// TIA Portal V20 export
FUNCTION_BLOCK "F-FB_Axis"   // FB130, F_LAD
{ S7_Optimized_Access := 'TRUE' }
// stored: AutoNumber false
   VAR
      LDrvSafe_SinaTlg903StatusAxis01_X : "LDrvSafe_SinaTlg903Status";
      LDrvSafe_SinaTlg903StatusAxis02_Y : "LDrvSafe_SinaTlg903Status";
      LDrvSafe_SinaTlg903StatusAxis03_ZM : "LDrvSafe_SinaTlg903Status";
      LDrvSafe_SinaTlg903StatusAxis04_B : "LDrvSafe_SinaTlg903Status";
      LDrvSafe_SinaTlg903StatusAxis05_U1 : "LDrvSafe_SinaTlg903Status";
      LDrvSafe_SinaTlg903StatusAxis06_U2 : "LDrvSafe_SinaTlg903Status";
      LDrvSafe_SinaTlg903StatusAxis07_V : "LDrvSafe_SinaTlg903Status";
      LDrvSafe_SinaTlg903StatusAxis08_W : "LDrvSafe_SinaTlg903Status";
      LDrvSafe_SinaTlg903StatusAxis09_ZL : "LDrvSafe_SinaTlg903Status";
      LDrvSafe_SinaTlg903ControlAxis01_X : "LDrvSafe_SinaTlg903Control";
      LDrvSafe_SinaTlg903ControlAxis02_Y : "LDrvSafe_SinaTlg903Control";
      LDrvSafe_SinaTlg903ControlAxis03_ZM : "LDrvSafe_SinaTlg903Control";
      LDrvSafe_SinaTlg903ControlAxis04_B : "LDrvSafe_SinaTlg903Control";
      LDrvSafe_SinaTlg903ControlAxis05_U1 : "LDrvSafe_SinaTlg903Control";
      LDrvSafe_SinaTlg903ControlAxis06_U2 : "LDrvSafe_SinaTlg903Control";
      LDrvSafe_SinaTlg903ControlAxis07_V : "LDrvSafe_SinaTlg903Control";
      LDrvSafe_SinaTlg903ControlAxis08_W : "LDrvSafe_SinaTlg903Control";
      LDrvSafe_SinaTlg903ControlAxis09_ZL : "LDrvSafe_SinaTlg903Control";
   END_VAR
   VAR_TEMP
      tEnable_Axis_Move : Bool;
   END_VAR
BEGIN

REGION Network 1: Enable Axis Move
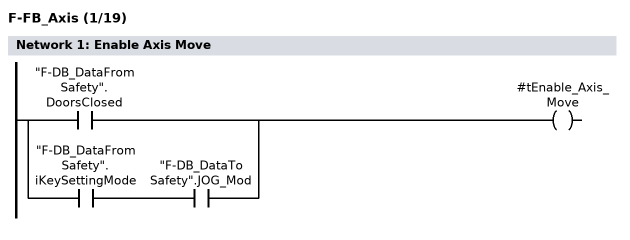
   RUNG wire#powerrail
      Contact( "F-DB_DataFromSafety".DoorsClosed )
      wire#w1
      Coil( #tEnable_Axis_Move )
   END_RUNG
   RUNG wire#powerrail
      Contact( "F-DB_DataFromSafety".iKeySettingMode )
      Contact( "F-DB_DataToSafety".JOG_Mod )
   END_RUNG wire#w1
   // the same network as SCL:
   #tEnable_Axis_Move := "F-DB_DataFromSafety".DoorsClosed OR ("F-DB_DataFromSafety".iKeySettingMode AND "F-DB_DataToSafety".JOG_Mod);
END_REGION

REGION Network 2: Axis01_X Status
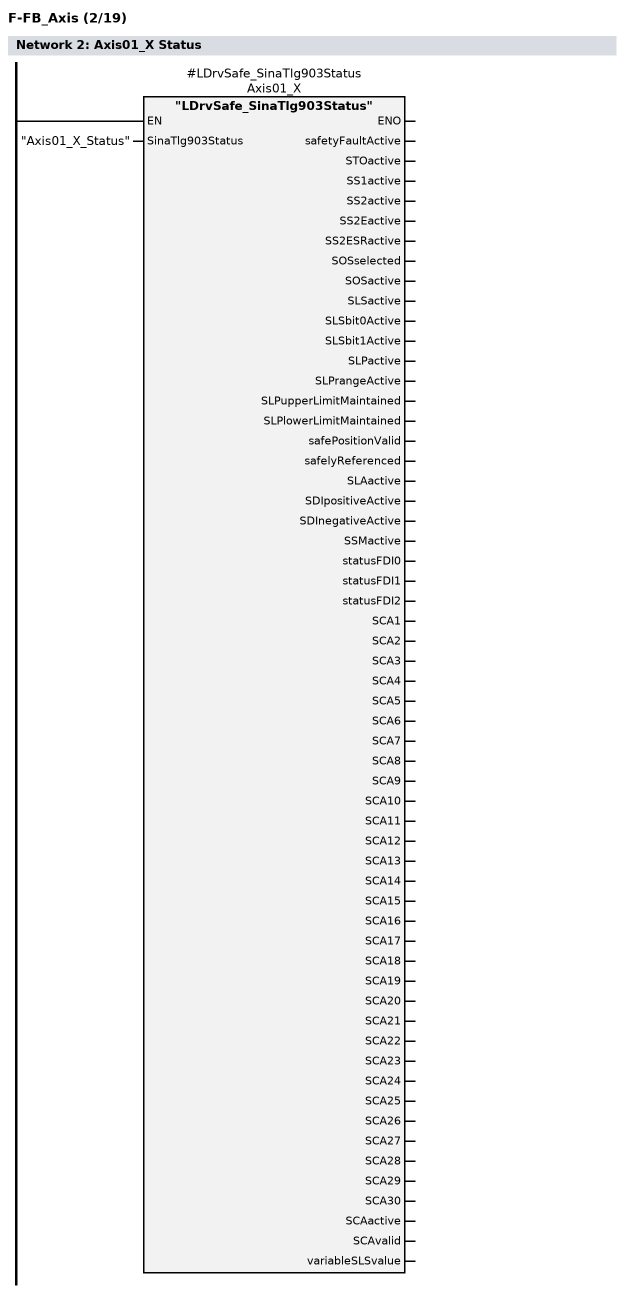
   RUNG wire#powerrail
      #LDrvSafe_SinaTlg903StatusAxis01_X(SinaTlg903Status := "Axis01_X_Status", safetyFaultActive =>, STOactive =>, SS1active =>, SS2active =>, SS2Eactive =>, SS2ESRactive =>, SOSselected =>, SOSactive =>, SLSactive =>, SLSbit0Active =>, SLSbit1Active =>, SLPactive =>, SLPrangeActive =>, SLPupperLimitMaintained =>, SLPlowerLimitMaintained =>, safePositionValid =>, safelyReferenced =>, SLAactive =>, SDIpositiveActive =>, SDInegativeActive =>, SSMactive =>, statusFDI0 =>, statusFDI1 =>, statusFDI2 =>, SCA1 =>, SCA2 =>, SCA3 =>, SCA4 =>, SCA5 =>, SCA6 =>, SCA7 =>, SCA8 =>, SCA9 =>, SCA10 =>, SCA11 =>, SCA12 =>, SCA13 =>, SCA14 =>, SCA15 =>, SCA16 =>, SCA17 =>, SCA18 =>, SCA19 =>, SCA20 =>, SCA21 =>, SCA22 =>, SCA23 =>, SCA24 =>, SCA25 =>, SCA26 =>, SCA27 =>, SCA28 =>, SCA29 =>, SCA30 =>, SCAactive =>, SCAvalid =>, variableSLSvalue =>)
   END_RUNG
   // the same network as SCL:
   #LDrvSafe_SinaTlg903StatusAxis01_X(SinaTlg903Status := "Axis01_X_Status");   // "LDrvSafe_SinaTlg903Status"
END_REGION

REGION Network 3: Axis01_X Control
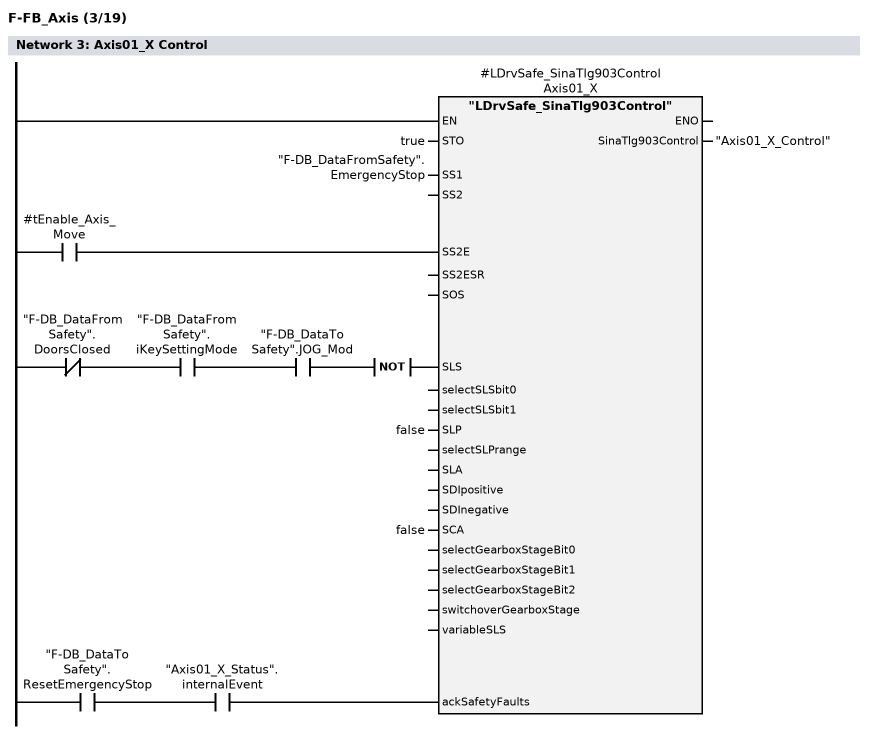
   RUNG wire#powerrail
      #LDrvSafe_SinaTlg903ControlAxis01_X(SS2E := wire#w1, SLS := wire#w2, ackSafetyFaults := wire#w3, STO := true, SS1 := "F-DB_DataFromSafety".EmergencyStop, SS2 :=, SS2ESR :=, SOS :=, selectSLSbit0 :=, selectSLSbit1 :=, SLP := false, selectSLPrange :=, SLA :=, SDIpositive :=, SDInegative :=, SCA := false, selectGearboxStageBit0 :=, selectGearboxStageBit1 :=, selectGearboxStageBit2 :=, switchoverGearboxStage :=, variableSLS :=, SinaTlg903Control => "Axis01_X_Control")
   END_RUNG
   RUNG wire#powerrail
      Contact( #tEnable_Axis_Move )
   END_RUNG wire#w1
   RUNG wire#powerrail
      I_Contact( "F-DB_DataFromSafety".DoorsClosed )
      Contact( "F-DB_DataFromSafety".iKeySettingMode )
      Contact( "F-DB_DataToSafety".JOG_Mod )
      Not()
   END_RUNG wire#w2
   RUNG wire#powerrail
      Contact( "F-DB_DataToSafety".ResetEmergencyStop )
      Contact( "Axis01_X_Status".internalEvent )
   END_RUNG wire#w3
   // the same network as SCL:
   #LDrvSafe_SinaTlg903ControlAxis01_X(STO := true,   // "LDrvSafe_SinaTlg903Control"
                           SS1 := "F-DB_DataFromSafety".EmergencyStop,
                           SS2E := #tEnable_Axis_Move,
                           SLS := NOT (NOT "F-DB_DataFromSafety".DoorsClosed AND "F-DB_DataFromSafety".iKeySettingMode AND "F-DB_DataToSafety".JOG_Mod),
                           SLP := false,
                           SCA := false,
                           ackSafetyFaults := "F-DB_DataToSafety".ResetEmergencyStop AND "Axis01_X_Status".internalEvent,
                           SinaTlg903Control => "Axis01_X_Control");
END_REGION

REGION Network 4: Axis02_Y Status
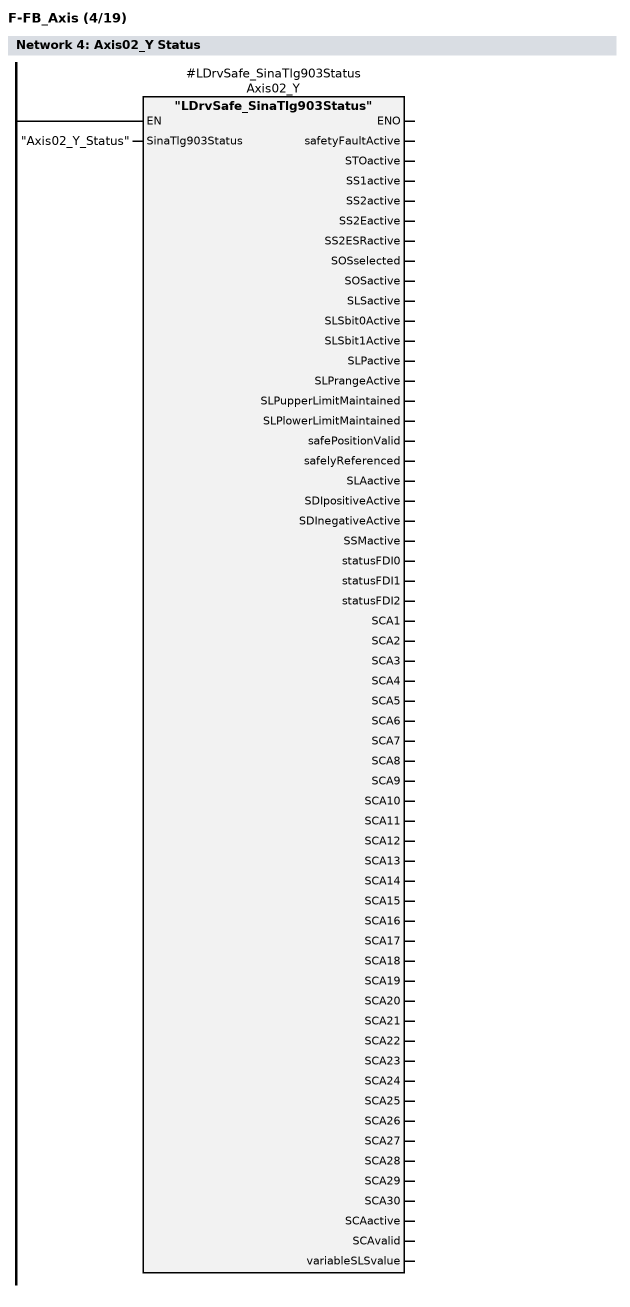
   RUNG wire#powerrail
      #LDrvSafe_SinaTlg903StatusAxis02_Y(SinaTlg903Status := "Axis02_Y_Status", safetyFaultActive =>, STOactive =>, SS1active =>, SS2active =>, SS2Eactive =>, SS2ESRactive =>, SOSselected =>, SOSactive =>, SLSactive =>, SLSbit0Active =>, SLSbit1Active =>, SLPactive =>, SLPrangeActive =>, SLPupperLimitMaintained =>, SLPlowerLimitMaintained =>, safePositionValid =>, safelyReferenced =>, SLAactive =>, SDIpositiveActive =>, SDInegativeActive =>, SSMactive =>, statusFDI0 =>, statusFDI1 =>, statusFDI2 =>, SCA1 =>, SCA2 =>, SCA3 =>, SCA4 =>, SCA5 =>, SCA6 =>, SCA7 =>, SCA8 =>, SCA9 =>, SCA10 =>, SCA11 =>, SCA12 =>, SCA13 =>, SCA14 =>, SCA15 =>, SCA16 =>, SCA17 =>, SCA18 =>, SCA19 =>, SCA20 =>, SCA21 =>, SCA22 =>, SCA23 =>, SCA24 =>, SCA25 =>, SCA26 =>, SCA27 =>, SCA28 =>, SCA29 =>, SCA30 =>, SCAactive =>, SCAvalid =>, variableSLSvalue =>)
   END_RUNG
   // the same network as SCL:
   #LDrvSafe_SinaTlg903StatusAxis02_Y(SinaTlg903Status := "Axis02_Y_Status");   // "LDrvSafe_SinaTlg903Status"
END_REGION

REGION Network 5: Axis02_Y Control
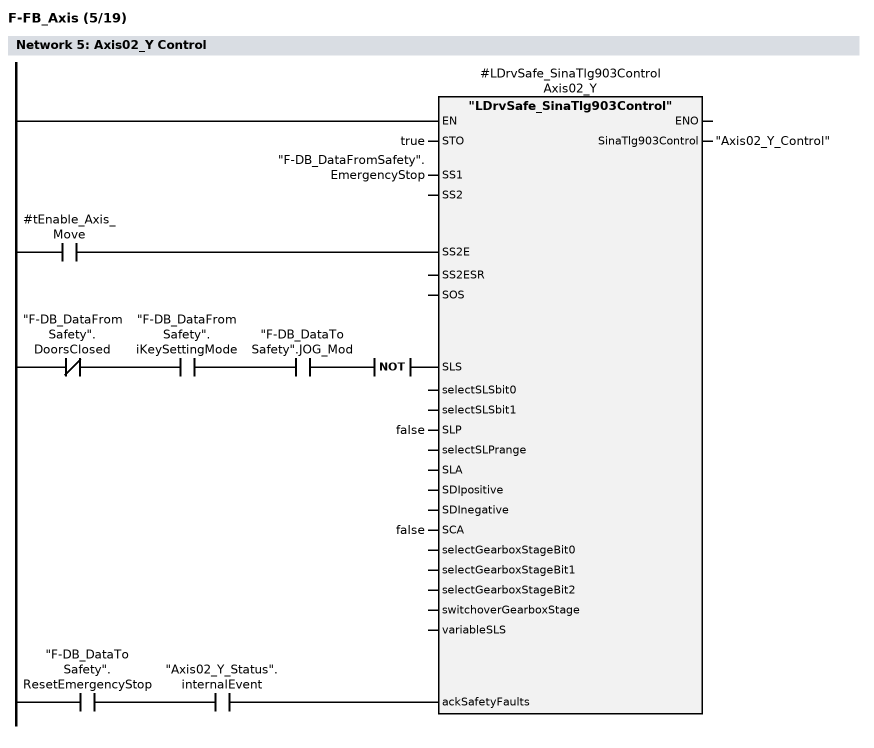
   RUNG wire#powerrail
      #LDrvSafe_SinaTlg903ControlAxis02_Y(SS2E := wire#w1, SLS := wire#w2, ackSafetyFaults := wire#w3, STO := true, SS1 := "F-DB_DataFromSafety".EmergencyStop, SS2 :=, SS2ESR :=, SOS :=, selectSLSbit0 :=, selectSLSbit1 :=, SLP := false, selectSLPrange :=, SLA :=, SDIpositive :=, SDInegative :=, SCA := false, selectGearboxStageBit0 :=, selectGearboxStageBit1 :=, selectGearboxStageBit2 :=, switchoverGearboxStage :=, variableSLS :=, SinaTlg903Control => "Axis02_Y_Control")
   END_RUNG
   RUNG wire#powerrail
      Contact( #tEnable_Axis_Move )
   END_RUNG wire#w1
   RUNG wire#powerrail
      I_Contact( "F-DB_DataFromSafety".DoorsClosed )
      Contact( "F-DB_DataFromSafety".iKeySettingMode )
      Contact( "F-DB_DataToSafety".JOG_Mod )
      Not()
   END_RUNG wire#w2
   RUNG wire#powerrail
      Contact( "F-DB_DataToSafety".ResetEmergencyStop )
      Contact( "Axis02_Y_Status".internalEvent )
   END_RUNG wire#w3
   // the same network as SCL:
   #LDrvSafe_SinaTlg903ControlAxis02_Y(STO := true,   // "LDrvSafe_SinaTlg903Control"
                           SS1 := "F-DB_DataFromSafety".EmergencyStop,
                           SS2E := #tEnable_Axis_Move,
                           SLS := NOT (NOT "F-DB_DataFromSafety".DoorsClosed AND "F-DB_DataFromSafety".iKeySettingMode AND "F-DB_DataToSafety".JOG_Mod),
                           SLP := false,
                           SCA := false,
                           ackSafetyFaults := "F-DB_DataToSafety".ResetEmergencyStop AND "Axis02_Y_Status".internalEvent,
                           SinaTlg903Control => "Axis02_Y_Control");
END_REGION

REGION Network 6: Axis03_ZM Status
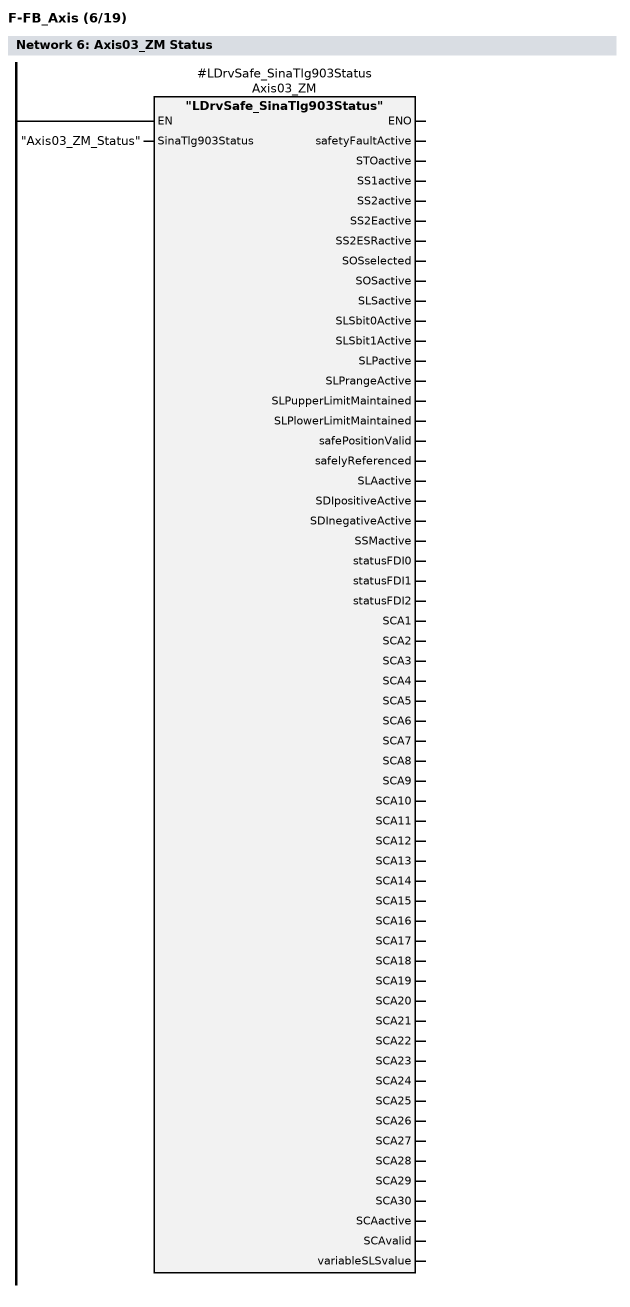
   RUNG wire#powerrail
      #LDrvSafe_SinaTlg903StatusAxis03_ZM(SinaTlg903Status := "Axis03_ZM_Status", safetyFaultActive =>, STOactive =>, SS1active =>, SS2active =>, SS2Eactive =>, SS2ESRactive =>, SOSselected =>, SOSactive =>, SLSactive =>, SLSbit0Active =>, SLSbit1Active =>, SLPactive =>, SLPrangeActive =>, SLPupperLimitMaintained =>, SLPlowerLimitMaintained =>, safePositionValid =>, safelyReferenced =>, SLAactive =>, SDIpositiveActive =>, SDInegativeActive =>, SSMactive =>, statusFDI0 =>, statusFDI1 =>, statusFDI2 =>, SCA1 =>, SCA2 =>, SCA3 =>, SCA4 =>, SCA5 =>, SCA6 =>, SCA7 =>, SCA8 =>, SCA9 =>, SCA10 =>, SCA11 =>, SCA12 =>, SCA13 =>, SCA14 =>, SCA15 =>, SCA16 =>, SCA17 =>, SCA18 =>, SCA19 =>, SCA20 =>, SCA21 =>, SCA22 =>, SCA23 =>, SCA24 =>, SCA25 =>, SCA26 =>, SCA27 =>, SCA28 =>, SCA29 =>, SCA30 =>, SCAactive =>, SCAvalid =>, variableSLSvalue =>)
   END_RUNG
   // the same network as SCL:
   #LDrvSafe_SinaTlg903StatusAxis03_ZM(SinaTlg903Status := "Axis03_ZM_Status");   // "LDrvSafe_SinaTlg903Status"
END_REGION

REGION Network 7: Axis03_ZM Control
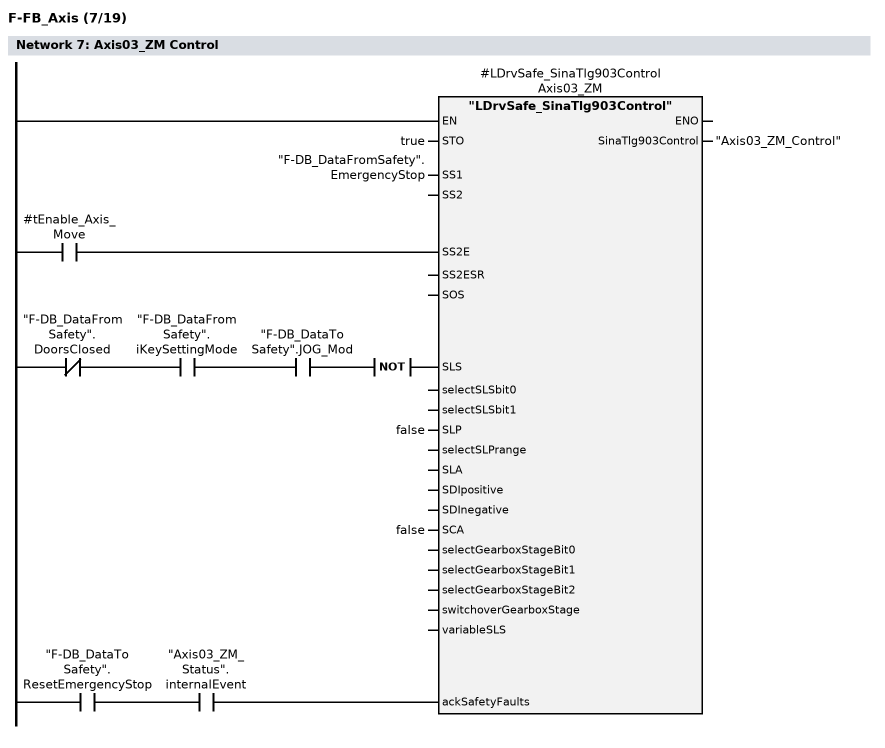
   RUNG wire#powerrail
      #LDrvSafe_SinaTlg903ControlAxis03_ZM(SS2E := wire#w1, SLS := wire#w2, ackSafetyFaults := wire#w3, STO := true, SS1 := "F-DB_DataFromSafety".EmergencyStop, SS2 :=, SS2ESR :=, SOS :=, selectSLSbit0 :=, selectSLSbit1 :=, SLP := false, selectSLPrange :=, SLA :=, SDIpositive :=, SDInegative :=, SCA := false, selectGearboxStageBit0 :=, selectGearboxStageBit1 :=, selectGearboxStageBit2 :=, switchoverGearboxStage :=, variableSLS :=, SinaTlg903Control => "Axis03_ZM_Control")
   END_RUNG
   RUNG wire#powerrail
      Contact( #tEnable_Axis_Move )
   END_RUNG wire#w1
   RUNG wire#powerrail
      I_Contact( "F-DB_DataFromSafety".DoorsClosed )
      Contact( "F-DB_DataFromSafety".iKeySettingMode )
      Contact( "F-DB_DataToSafety".JOG_Mod )
      Not()
   END_RUNG wire#w2
   RUNG wire#powerrail
      Contact( "F-DB_DataToSafety".ResetEmergencyStop )
      Contact( "Axis03_ZM_Status".internalEvent )
   END_RUNG wire#w3
   // the same network as SCL:
   #LDrvSafe_SinaTlg903ControlAxis03_ZM(STO := true,   // "LDrvSafe_SinaTlg903Control"
                           SS1 := "F-DB_DataFromSafety".EmergencyStop,
                           SS2E := #tEnable_Axis_Move,
                           SLS := NOT (NOT "F-DB_DataFromSafety".DoorsClosed AND "F-DB_DataFromSafety".iKeySettingMode AND "F-DB_DataToSafety".JOG_Mod),
                           SLP := false,
                           SCA := false,
                           ackSafetyFaults := "F-DB_DataToSafety".ResetEmergencyStop AND "Axis03_ZM_Status".internalEvent,
                           SinaTlg903Control => "Axis03_ZM_Control");
END_REGION

REGION Network 8: Axis04_B Status
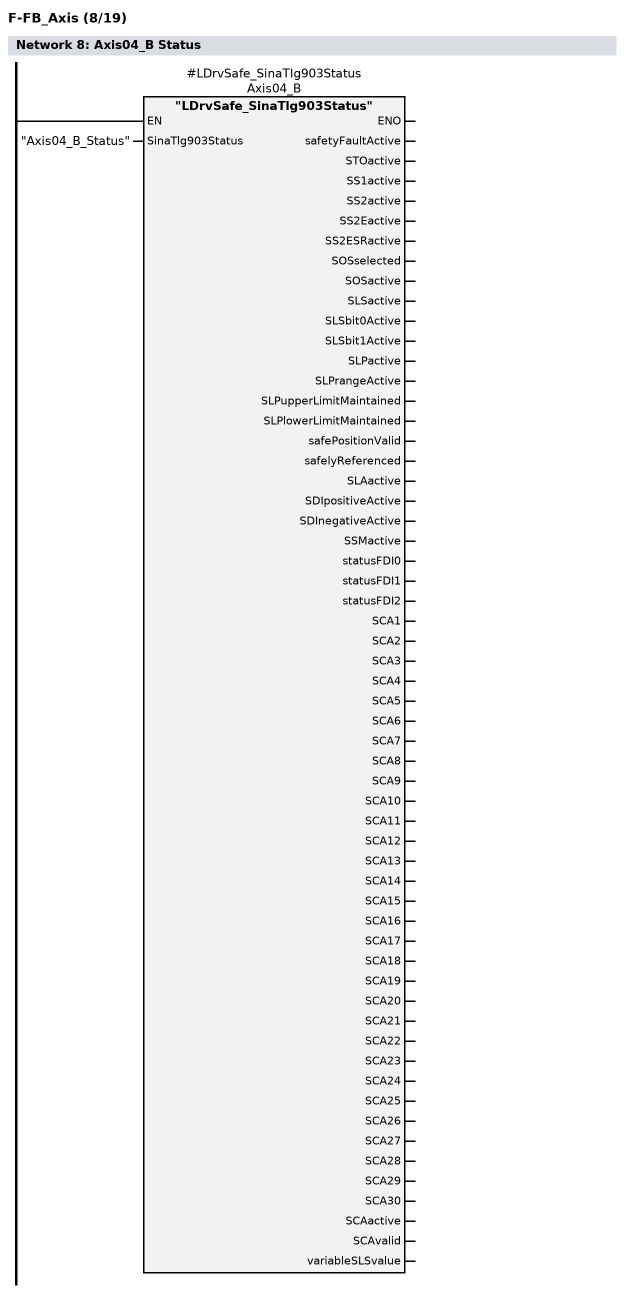
   RUNG wire#powerrail
      #LDrvSafe_SinaTlg903StatusAxis04_B(SinaTlg903Status := "Axis04_B_Status", safetyFaultActive =>, STOactive =>, SS1active =>, SS2active =>, SS2Eactive =>, SS2ESRactive =>, SOSselected =>, SOSactive =>, SLSactive =>, SLSbit0Active =>, SLSbit1Active =>, SLPactive =>, SLPrangeActive =>, SLPupperLimitMaintained =>, SLPlowerLimitMaintained =>, safePositionValid =>, safelyReferenced =>, SLAactive =>, SDIpositiveActive =>, SDInegativeActive =>, SSMactive =>, statusFDI0 =>, statusFDI1 =>, statusFDI2 =>, SCA1 =>, SCA2 =>, SCA3 =>, SCA4 =>, SCA5 =>, SCA6 =>, SCA7 =>, SCA8 =>, SCA9 =>, SCA10 =>, SCA11 =>, SCA12 =>, SCA13 =>, SCA14 =>, SCA15 =>, SCA16 =>, SCA17 =>, SCA18 =>, SCA19 =>, SCA20 =>, SCA21 =>, SCA22 =>, SCA23 =>, SCA24 =>, SCA25 =>, SCA26 =>, SCA27 =>, SCA28 =>, SCA29 =>, SCA30 =>, SCAactive =>, SCAvalid =>, variableSLSvalue =>)
   END_RUNG
   // the same network as SCL:
   #LDrvSafe_SinaTlg903StatusAxis04_B(SinaTlg903Status := "Axis04_B_Status");   // "LDrvSafe_SinaTlg903Status"
END_REGION

REGION Network 9: Axis04_B Control
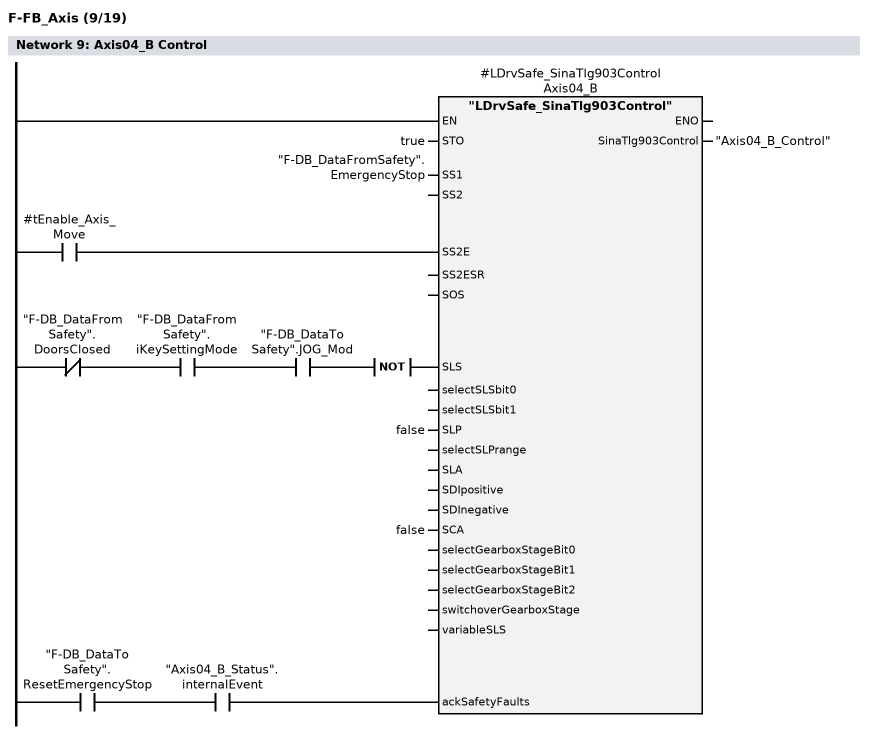
   RUNG wire#powerrail
      #LDrvSafe_SinaTlg903ControlAxis04_B(SS2E := wire#w1, SLS := wire#w2, ackSafetyFaults := wire#w3, STO := true, SS1 := "F-DB_DataFromSafety".EmergencyStop, SS2 :=, SS2ESR :=, SOS :=, selectSLSbit0 :=, selectSLSbit1 :=, SLP := false, selectSLPrange :=, SLA :=, SDIpositive :=, SDInegative :=, SCA := false, selectGearboxStageBit0 :=, selectGearboxStageBit1 :=, selectGearboxStageBit2 :=, switchoverGearboxStage :=, variableSLS :=, SinaTlg903Control => "Axis04_B_Control")
   END_RUNG
   RUNG wire#powerrail
      Contact( #tEnable_Axis_Move )
   END_RUNG wire#w1
   RUNG wire#powerrail
      I_Contact( "F-DB_DataFromSafety".DoorsClosed )
      Contact( "F-DB_DataFromSafety".iKeySettingMode )
      Contact( "F-DB_DataToSafety".JOG_Mod )
      Not()
   END_RUNG wire#w2
   RUNG wire#powerrail
      Contact( "F-DB_DataToSafety".ResetEmergencyStop )
      Contact( "Axis04_B_Status".internalEvent )
   END_RUNG wire#w3
   // the same network as SCL:
   #LDrvSafe_SinaTlg903ControlAxis04_B(STO := true,   // "LDrvSafe_SinaTlg903Control"
                           SS1 := "F-DB_DataFromSafety".EmergencyStop,
                           SS2E := #tEnable_Axis_Move,
                           SLS := NOT (NOT "F-DB_DataFromSafety".DoorsClosed AND "F-DB_DataFromSafety".iKeySettingMode AND "F-DB_DataToSafety".JOG_Mod),
                           SLP := false,
                           SCA := false,
                           ackSafetyFaults := "F-DB_DataToSafety".ResetEmergencyStop AND "Axis04_B_Status".internalEvent,
                           SinaTlg903Control => "Axis04_B_Control");
END_REGION

REGION Network 10: Axis05_U1 Status
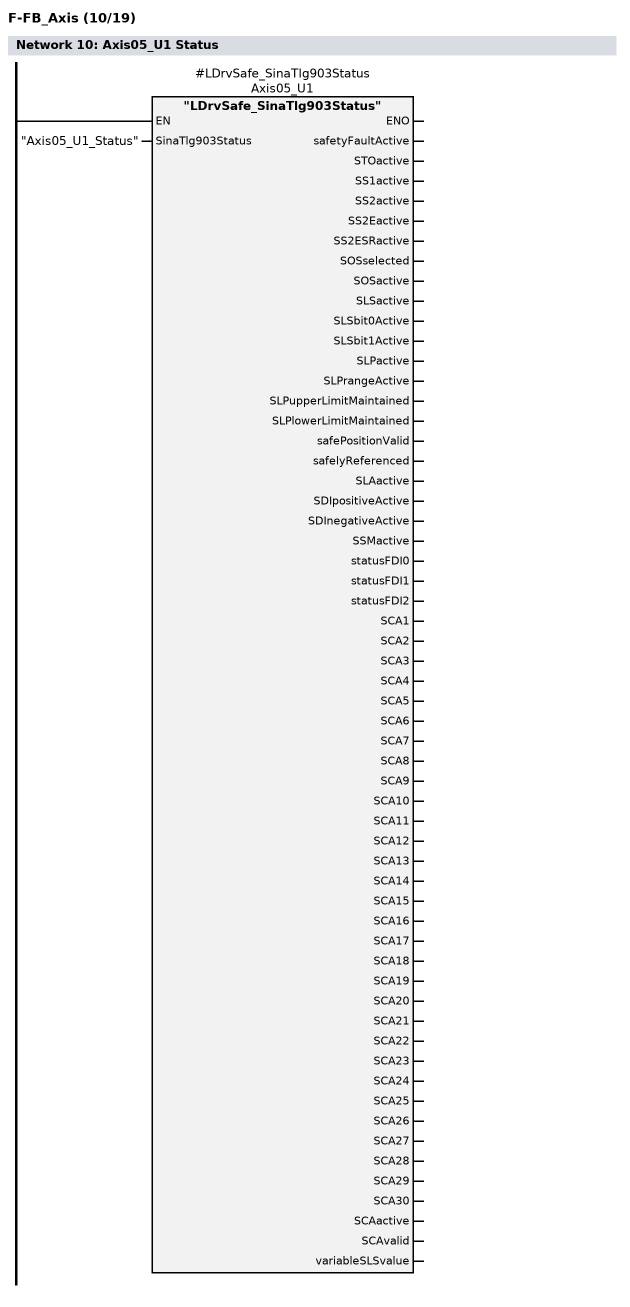
   RUNG wire#powerrail
      #LDrvSafe_SinaTlg903StatusAxis05_U1(SinaTlg903Status := "Axis05_U1_Status", safetyFaultActive =>, STOactive =>, SS1active =>, SS2active =>, SS2Eactive =>, SS2ESRactive =>, SOSselected =>, SOSactive =>, SLSactive =>, SLSbit0Active =>, SLSbit1Active =>, SLPactive =>, SLPrangeActive =>, SLPupperLimitMaintained =>, SLPlowerLimitMaintained =>, safePositionValid =>, safelyReferenced =>, SLAactive =>, SDIpositiveActive =>, SDInegativeActive =>, SSMactive =>, statusFDI0 =>, statusFDI1 =>, statusFDI2 =>, SCA1 =>, SCA2 =>, SCA3 =>, SCA4 =>, SCA5 =>, SCA6 =>, SCA7 =>, SCA8 =>, SCA9 =>, SCA10 =>, SCA11 =>, SCA12 =>, SCA13 =>, SCA14 =>, SCA15 =>, SCA16 =>, SCA17 =>, SCA18 =>, SCA19 =>, SCA20 =>, SCA21 =>, SCA22 =>, SCA23 =>, SCA24 =>, SCA25 =>, SCA26 =>, SCA27 =>, SCA28 =>, SCA29 =>, SCA30 =>, SCAactive =>, SCAvalid =>, variableSLSvalue =>)
   END_RUNG
   // the same network as SCL:
   #LDrvSafe_SinaTlg903StatusAxis05_U1(SinaTlg903Status := "Axis05_U1_Status");   // "LDrvSafe_SinaTlg903Status"
END_REGION

REGION Network 11: Axis05_U1 Control
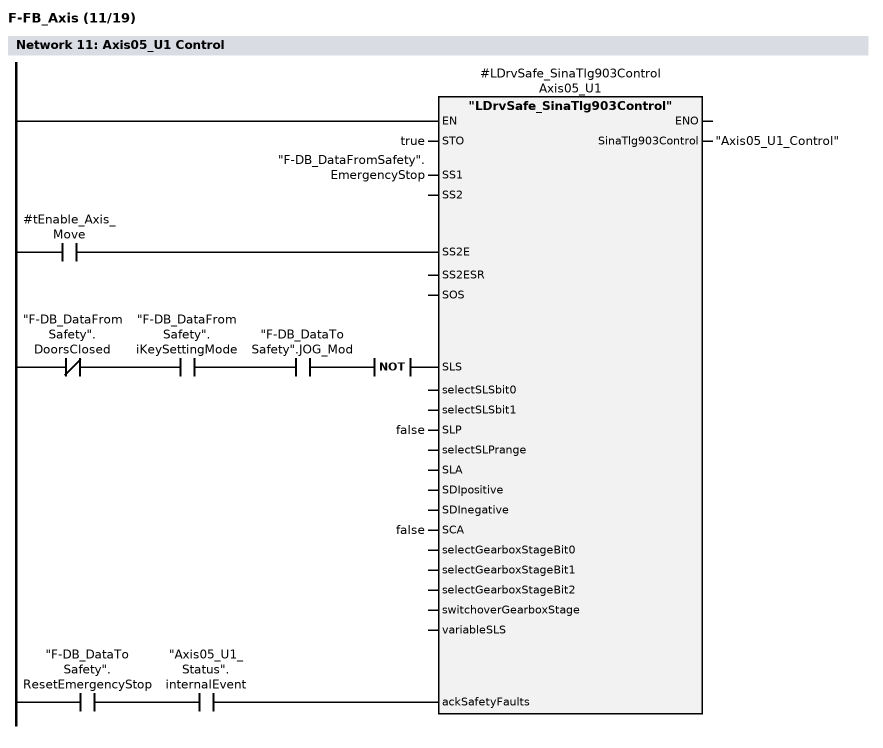
   RUNG wire#powerrail
      #LDrvSafe_SinaTlg903ControlAxis05_U1(SS2E := wire#w1, SLS := wire#w2, ackSafetyFaults := wire#w3, STO := true, SS1 := "F-DB_DataFromSafety".EmergencyStop, SS2 :=, SS2ESR :=, SOS :=, selectSLSbit0 :=, selectSLSbit1 :=, SLP := false, selectSLPrange :=, SLA :=, SDIpositive :=, SDInegative :=, SCA := false, selectGearboxStageBit0 :=, selectGearboxStageBit1 :=, selectGearboxStageBit2 :=, switchoverGearboxStage :=, variableSLS :=, SinaTlg903Control => "Axis05_U1_Control")
   END_RUNG
   RUNG wire#powerrail
      Contact( #tEnable_Axis_Move )
   END_RUNG wire#w1
   RUNG wire#powerrail
      I_Contact( "F-DB_DataFromSafety".DoorsClosed )
      Contact( "F-DB_DataFromSafety".iKeySettingMode )
      Contact( "F-DB_DataToSafety".JOG_Mod )
      Not()
   END_RUNG wire#w2
   RUNG wire#powerrail
      Contact( "F-DB_DataToSafety".ResetEmergencyStop )
      Contact( "Axis05_U1_Status".internalEvent )
   END_RUNG wire#w3
   // the same network as SCL:
   #LDrvSafe_SinaTlg903ControlAxis05_U1(STO := true,   // "LDrvSafe_SinaTlg903Control"
                           SS1 := "F-DB_DataFromSafety".EmergencyStop,
                           SS2E := #tEnable_Axis_Move,
                           SLS := NOT (NOT "F-DB_DataFromSafety".DoorsClosed AND "F-DB_DataFromSafety".iKeySettingMode AND "F-DB_DataToSafety".JOG_Mod),
                           SLP := false,
                           SCA := false,
                           ackSafetyFaults := "F-DB_DataToSafety".ResetEmergencyStop AND "Axis05_U1_Status".internalEvent,
                           SinaTlg903Control => "Axis05_U1_Control");
END_REGION

REGION Network 12: Axis06_U2 Status
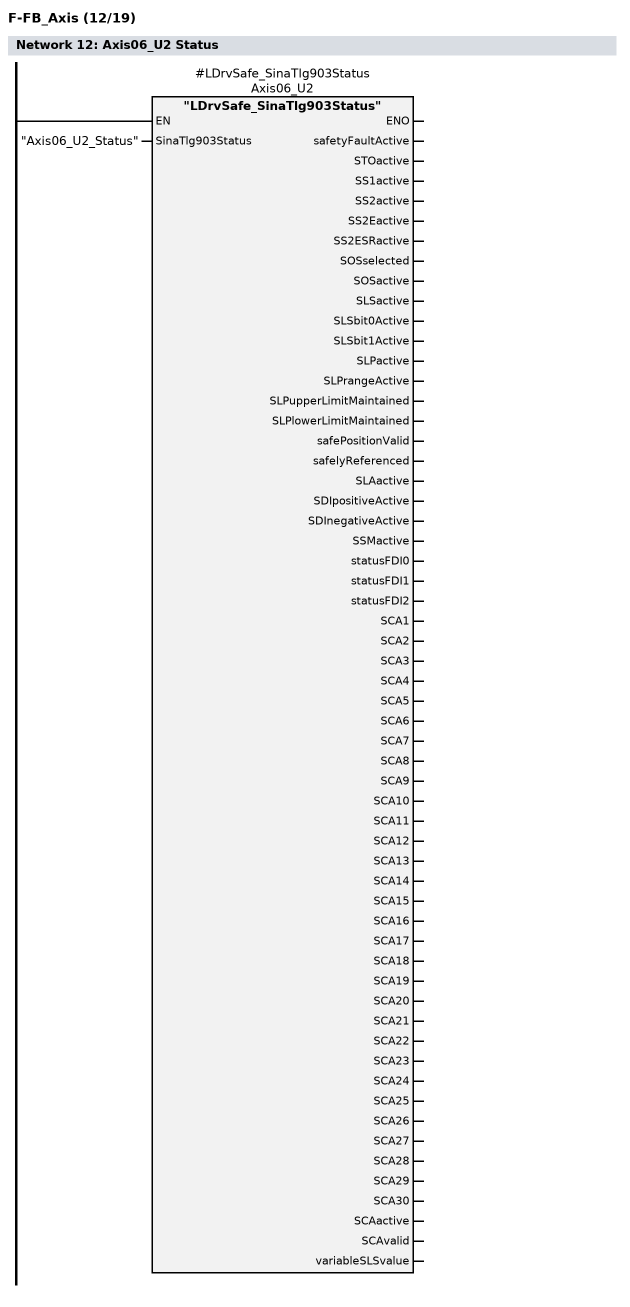
   RUNG wire#powerrail
      #LDrvSafe_SinaTlg903StatusAxis06_U2(SinaTlg903Status := "Axis06_U2_Status", safetyFaultActive =>, STOactive =>, SS1active =>, SS2active =>, SS2Eactive =>, SS2ESRactive =>, SOSselected =>, SOSactive =>, SLSactive =>, SLSbit0Active =>, SLSbit1Active =>, SLPactive =>, SLPrangeActive =>, SLPupperLimitMaintained =>, SLPlowerLimitMaintained =>, safePositionValid =>, safelyReferenced =>, SLAactive =>, SDIpositiveActive =>, SDInegativeActive =>, SSMactive =>, statusFDI0 =>, statusFDI1 =>, statusFDI2 =>, SCA1 =>, SCA2 =>, SCA3 =>, SCA4 =>, SCA5 =>, SCA6 =>, SCA7 =>, SCA8 =>, SCA9 =>, SCA10 =>, SCA11 =>, SCA12 =>, SCA13 =>, SCA14 =>, SCA15 =>, SCA16 =>, SCA17 =>, SCA18 =>, SCA19 =>, SCA20 =>, SCA21 =>, SCA22 =>, SCA23 =>, SCA24 =>, SCA25 =>, SCA26 =>, SCA27 =>, SCA28 =>, SCA29 =>, SCA30 =>, SCAactive =>, SCAvalid =>, variableSLSvalue =>)
   END_RUNG
   // the same network as SCL:
   #LDrvSafe_SinaTlg903StatusAxis06_U2(SinaTlg903Status := "Axis06_U2_Status");   // "LDrvSafe_SinaTlg903Status"
END_REGION

REGION Network 13: Axis06_U2 Control
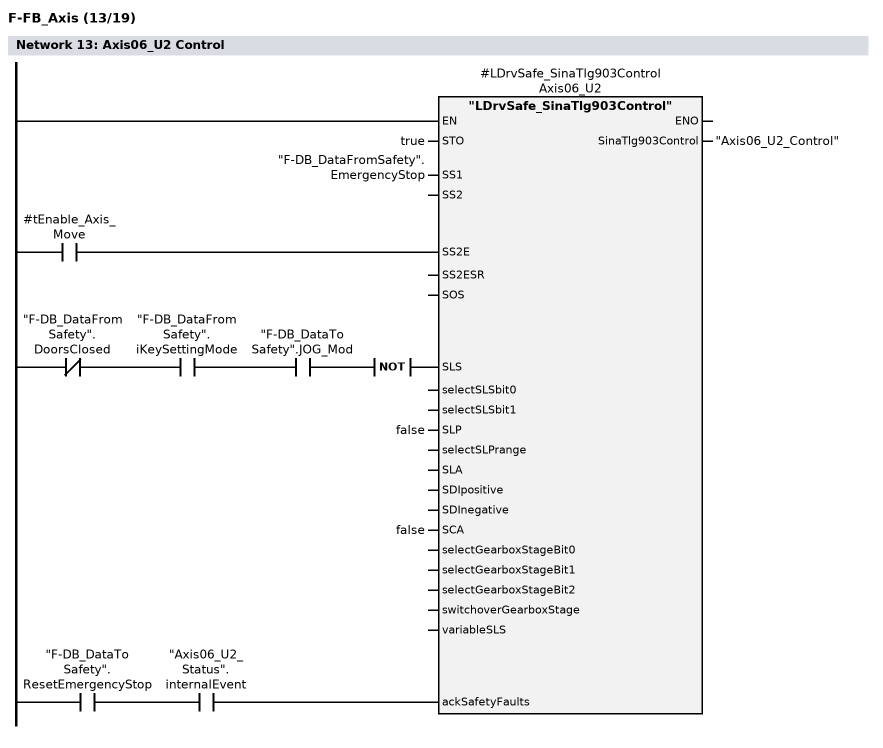
   RUNG wire#powerrail
      #LDrvSafe_SinaTlg903ControlAxis06_U2(SS2E := wire#w1, SLS := wire#w2, ackSafetyFaults := wire#w3, STO := true, SS1 := "F-DB_DataFromSafety".EmergencyStop, SS2 :=, SS2ESR :=, SOS :=, selectSLSbit0 :=, selectSLSbit1 :=, SLP := false, selectSLPrange :=, SLA :=, SDIpositive :=, SDInegative :=, SCA := false, selectGearboxStageBit0 :=, selectGearboxStageBit1 :=, selectGearboxStageBit2 :=, switchoverGearboxStage :=, variableSLS :=, SinaTlg903Control => "Axis06_U2_Control")
   END_RUNG
   RUNG wire#powerrail
      Contact( #tEnable_Axis_Move )
   END_RUNG wire#w1
   RUNG wire#powerrail
      I_Contact( "F-DB_DataFromSafety".DoorsClosed )
      Contact( "F-DB_DataFromSafety".iKeySettingMode )
      Contact( "F-DB_DataToSafety".JOG_Mod )
      Not()
   END_RUNG wire#w2
   RUNG wire#powerrail
      Contact( "F-DB_DataToSafety".ResetEmergencyStop )
      Contact( "Axis06_U2_Status".internalEvent )
   END_RUNG wire#w3
   // the same network as SCL:
   #LDrvSafe_SinaTlg903ControlAxis06_U2(STO := true,   // "LDrvSafe_SinaTlg903Control"
                           SS1 := "F-DB_DataFromSafety".EmergencyStop,
                           SS2E := #tEnable_Axis_Move,
                           SLS := NOT (NOT "F-DB_DataFromSafety".DoorsClosed AND "F-DB_DataFromSafety".iKeySettingMode AND "F-DB_DataToSafety".JOG_Mod),
                           SLP := false,
                           SCA := false,
                           ackSafetyFaults := "F-DB_DataToSafety".ResetEmergencyStop AND "Axis06_U2_Status".internalEvent,
                           SinaTlg903Control => "Axis06_U2_Control");
END_REGION

REGION Network 14: Axis07_V Status
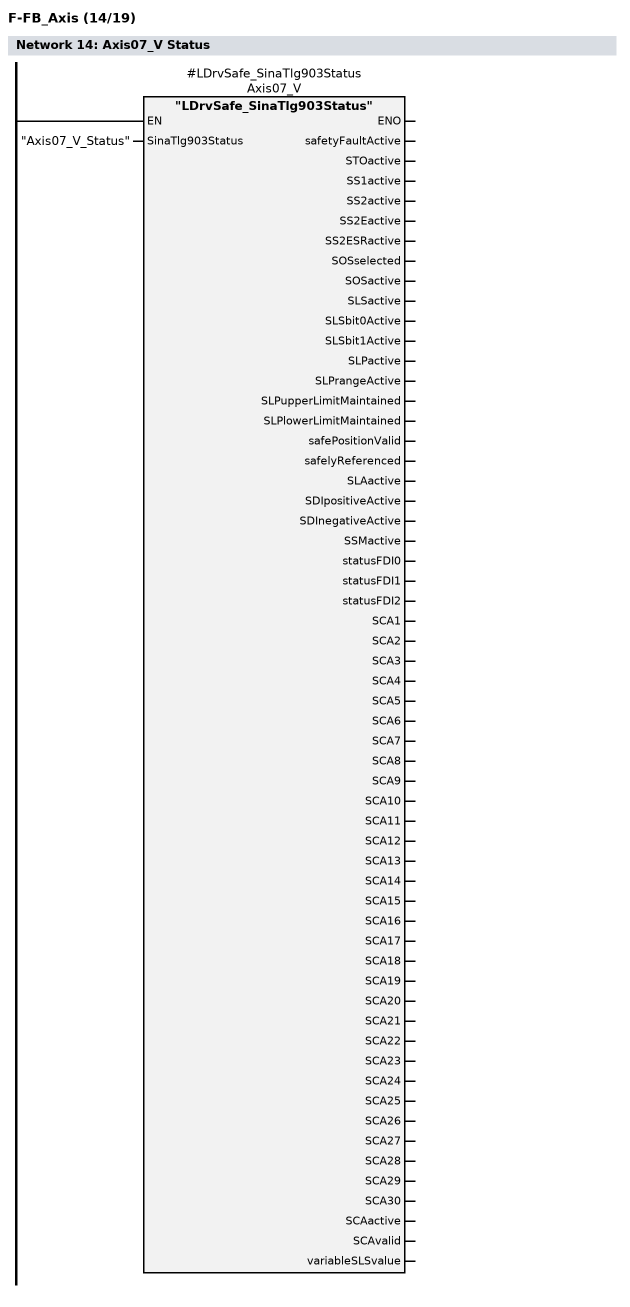
   RUNG wire#powerrail
      #LDrvSafe_SinaTlg903StatusAxis07_V(SinaTlg903Status := "Axis07_V_Status", safetyFaultActive =>, STOactive =>, SS1active =>, SS2active =>, SS2Eactive =>, SS2ESRactive =>, SOSselected =>, SOSactive =>, SLSactive =>, SLSbit0Active =>, SLSbit1Active =>, SLPactive =>, SLPrangeActive =>, SLPupperLimitMaintained =>, SLPlowerLimitMaintained =>, safePositionValid =>, safelyReferenced =>, SLAactive =>, SDIpositiveActive =>, SDInegativeActive =>, SSMactive =>, statusFDI0 =>, statusFDI1 =>, statusFDI2 =>, SCA1 =>, SCA2 =>, SCA3 =>, SCA4 =>, SCA5 =>, SCA6 =>, SCA7 =>, SCA8 =>, SCA9 =>, SCA10 =>, SCA11 =>, SCA12 =>, SCA13 =>, SCA14 =>, SCA15 =>, SCA16 =>, SCA17 =>, SCA18 =>, SCA19 =>, SCA20 =>, SCA21 =>, SCA22 =>, SCA23 =>, SCA24 =>, SCA25 =>, SCA26 =>, SCA27 =>, SCA28 =>, SCA29 =>, SCA30 =>, SCAactive =>, SCAvalid =>, variableSLSvalue =>)
   END_RUNG
   // the same network as SCL:
   #LDrvSafe_SinaTlg903StatusAxis07_V(SinaTlg903Status := "Axis07_V_Status");   // "LDrvSafe_SinaTlg903Status"
END_REGION

REGION Network 15: Axis07_V Control
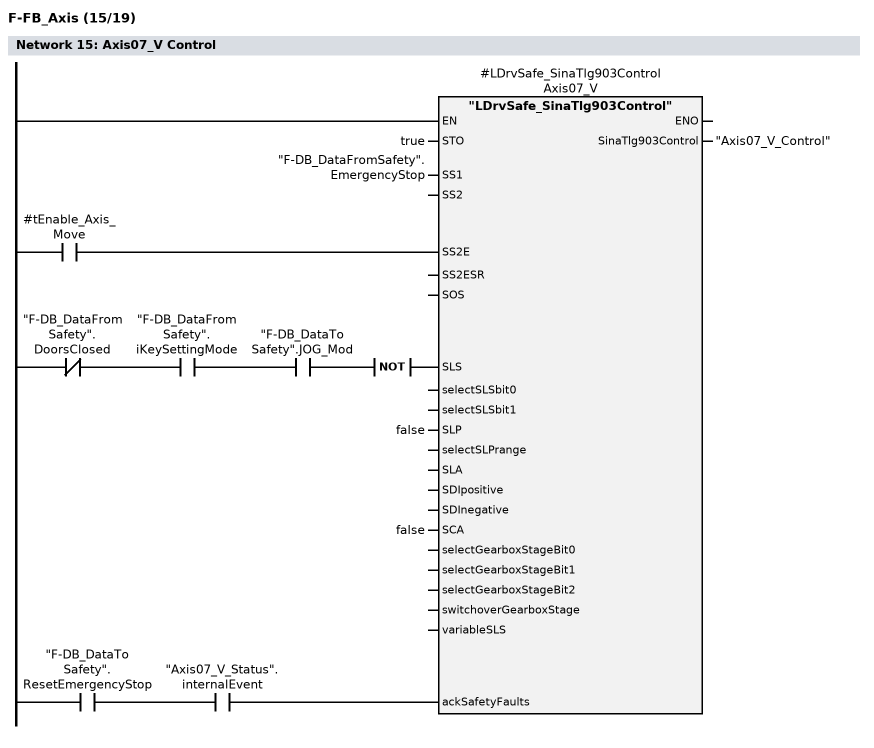
   RUNG wire#powerrail
      #LDrvSafe_SinaTlg903ControlAxis07_V(SS2E := wire#w1, SLS := wire#w2, ackSafetyFaults := wire#w3, STO := true, SS1 := "F-DB_DataFromSafety".EmergencyStop, SS2 :=, SS2ESR :=, SOS :=, selectSLSbit0 :=, selectSLSbit1 :=, SLP := false, selectSLPrange :=, SLA :=, SDIpositive :=, SDInegative :=, SCA := false, selectGearboxStageBit0 :=, selectGearboxStageBit1 :=, selectGearboxStageBit2 :=, switchoverGearboxStage :=, variableSLS :=, SinaTlg903Control => "Axis07_V_Control")
   END_RUNG
   RUNG wire#powerrail
      Contact( #tEnable_Axis_Move )
   END_RUNG wire#w1
   RUNG wire#powerrail
      I_Contact( "F-DB_DataFromSafety".DoorsClosed )
      Contact( "F-DB_DataFromSafety".iKeySettingMode )
      Contact( "F-DB_DataToSafety".JOG_Mod )
      Not()
   END_RUNG wire#w2
   RUNG wire#powerrail
      Contact( "F-DB_DataToSafety".ResetEmergencyStop )
      Contact( "Axis07_V_Status".internalEvent )
   END_RUNG wire#w3
   // the same network as SCL:
   #LDrvSafe_SinaTlg903ControlAxis07_V(STO := true,   // "LDrvSafe_SinaTlg903Control"
                           SS1 := "F-DB_DataFromSafety".EmergencyStop,
                           SS2E := #tEnable_Axis_Move,
                           SLS := NOT (NOT "F-DB_DataFromSafety".DoorsClosed AND "F-DB_DataFromSafety".iKeySettingMode AND "F-DB_DataToSafety".JOG_Mod),
                           SLP := false,
                           SCA := false,
                           ackSafetyFaults := "F-DB_DataToSafety".ResetEmergencyStop AND "Axis07_V_Status".internalEvent,
                           SinaTlg903Control => "Axis07_V_Control");
END_REGION

REGION Network 16: Axis08_W Status
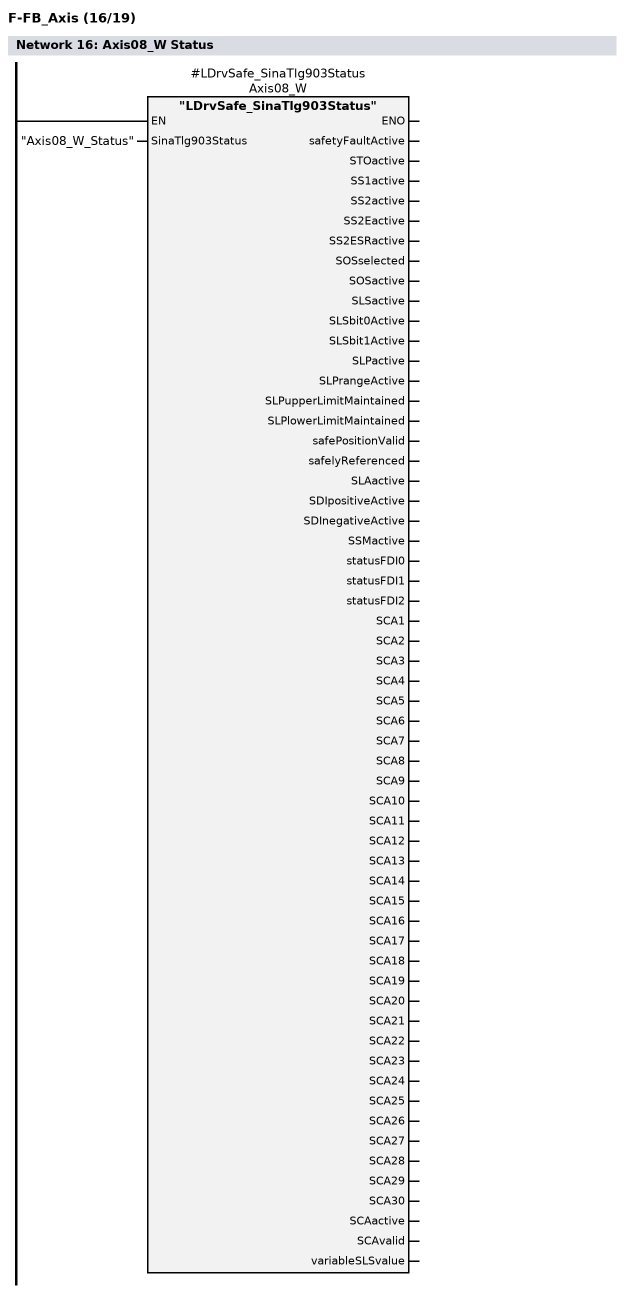
   RUNG wire#powerrail
      #LDrvSafe_SinaTlg903StatusAxis08_W(SinaTlg903Status := "Axis08_W_Status", safetyFaultActive =>, STOactive =>, SS1active =>, SS2active =>, SS2Eactive =>, SS2ESRactive =>, SOSselected =>, SOSactive =>, SLSactive =>, SLSbit0Active =>, SLSbit1Active =>, SLPactive =>, SLPrangeActive =>, SLPupperLimitMaintained =>, SLPlowerLimitMaintained =>, safePositionValid =>, safelyReferenced =>, SLAactive =>, SDIpositiveActive =>, SDInegativeActive =>, SSMactive =>, statusFDI0 =>, statusFDI1 =>, statusFDI2 =>, SCA1 =>, SCA2 =>, SCA3 =>, SCA4 =>, SCA5 =>, SCA6 =>, SCA7 =>, SCA8 =>, SCA9 =>, SCA10 =>, SCA11 =>, SCA12 =>, SCA13 =>, SCA14 =>, SCA15 =>, SCA16 =>, SCA17 =>, SCA18 =>, SCA19 =>, SCA20 =>, SCA21 =>, SCA22 =>, SCA23 =>, SCA24 =>, SCA25 =>, SCA26 =>, SCA27 =>, SCA28 =>, SCA29 =>, SCA30 =>, SCAactive =>, SCAvalid =>, variableSLSvalue =>)
   END_RUNG
   // the same network as SCL:
   #LDrvSafe_SinaTlg903StatusAxis08_W(SinaTlg903Status := "Axis08_W_Status");   // "LDrvSafe_SinaTlg903Status"
END_REGION

REGION Network 17: Axis08_W Control
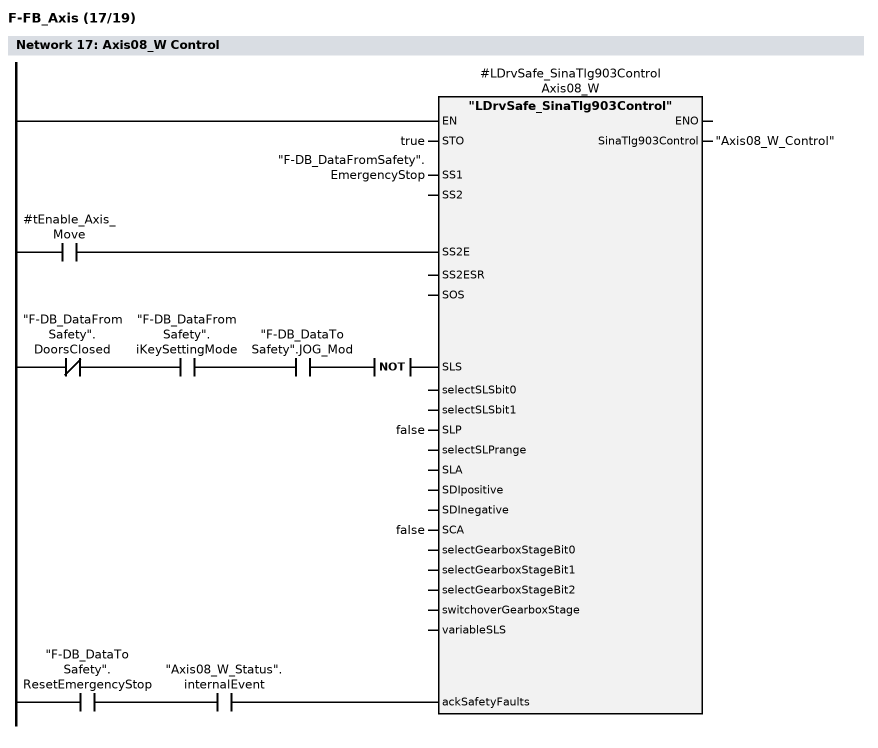
   RUNG wire#powerrail
      #LDrvSafe_SinaTlg903ControlAxis08_W(SS2E := wire#w1, SLS := wire#w2, ackSafetyFaults := wire#w3, STO := true, SS1 := "F-DB_DataFromSafety".EmergencyStop, SS2 :=, SS2ESR :=, SOS :=, selectSLSbit0 :=, selectSLSbit1 :=, SLP := false, selectSLPrange :=, SLA :=, SDIpositive :=, SDInegative :=, SCA := false, selectGearboxStageBit0 :=, selectGearboxStageBit1 :=, selectGearboxStageBit2 :=, switchoverGearboxStage :=, variableSLS :=, SinaTlg903Control => "Axis08_W_Control")
   END_RUNG
   RUNG wire#powerrail
      Contact( #tEnable_Axis_Move )
   END_RUNG wire#w1
   RUNG wire#powerrail
      I_Contact( "F-DB_DataFromSafety".DoorsClosed )
      Contact( "F-DB_DataFromSafety".iKeySettingMode )
      Contact( "F-DB_DataToSafety".JOG_Mod )
      Not()
   END_RUNG wire#w2
   RUNG wire#powerrail
      Contact( "F-DB_DataToSafety".ResetEmergencyStop )
      Contact( "Axis08_W_Status".internalEvent )
   END_RUNG wire#w3
   // the same network as SCL:
   #LDrvSafe_SinaTlg903ControlAxis08_W(STO := true,   // "LDrvSafe_SinaTlg903Control"
                           SS1 := "F-DB_DataFromSafety".EmergencyStop,
                           SS2E := #tEnable_Axis_Move,
                           SLS := NOT (NOT "F-DB_DataFromSafety".DoorsClosed AND "F-DB_DataFromSafety".iKeySettingMode AND "F-DB_DataToSafety".JOG_Mod),
                           SLP := false,
                           SCA := false,
                           ackSafetyFaults := "F-DB_DataToSafety".ResetEmergencyStop AND "Axis08_W_Status".internalEvent,
                           SinaTlg903Control => "Axis08_W_Control");
END_REGION

REGION Network 18: Axis09_ZL Status
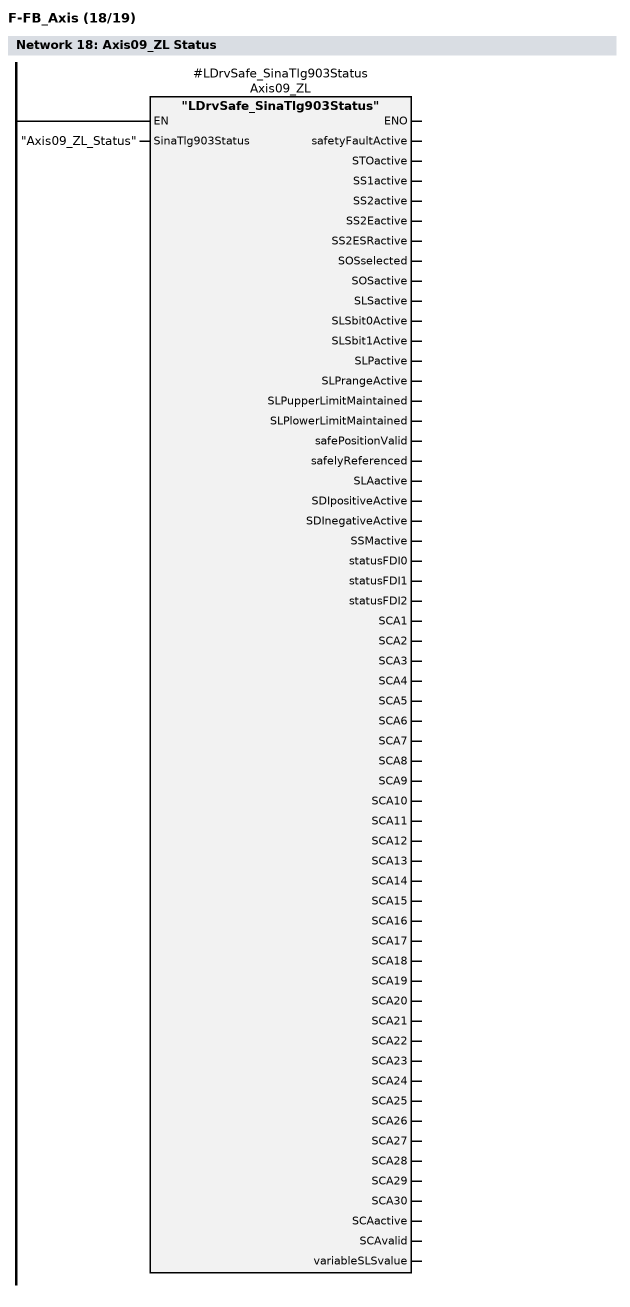
   RUNG wire#powerrail
      #LDrvSafe_SinaTlg903StatusAxis09_ZL(SinaTlg903Status := "Axis09_ZL_Status", safetyFaultActive =>, STOactive =>, SS1active =>, SS2active =>, SS2Eactive =>, SS2ESRactive =>, SOSselected =>, SOSactive =>, SLSactive =>, SLSbit0Active =>, SLSbit1Active =>, SLPactive =>, SLPrangeActive =>, SLPupperLimitMaintained =>, SLPlowerLimitMaintained =>, safePositionValid =>, safelyReferenced =>, SLAactive =>, SDIpositiveActive =>, SDInegativeActive =>, SSMactive =>, statusFDI0 =>, statusFDI1 =>, statusFDI2 =>, SCA1 =>, SCA2 =>, SCA3 =>, SCA4 =>, SCA5 =>, SCA6 =>, SCA7 =>, SCA8 =>, SCA9 =>, SCA10 =>, SCA11 =>, SCA12 =>, SCA13 =>, SCA14 =>, SCA15 =>, SCA16 =>, SCA17 =>, SCA18 =>, SCA19 =>, SCA20 =>, SCA21 =>, SCA22 =>, SCA23 =>, SCA24 =>, SCA25 =>, SCA26 =>, SCA27 =>, SCA28 =>, SCA29 =>, SCA30 =>, SCAactive =>, SCAvalid =>, variableSLSvalue =>)
   END_RUNG
   // the same network as SCL:
   #LDrvSafe_SinaTlg903StatusAxis09_ZL(SinaTlg903Status := "Axis09_ZL_Status");   // "LDrvSafe_SinaTlg903Status"
END_REGION

REGION Network 19: Axis09_ZL Control
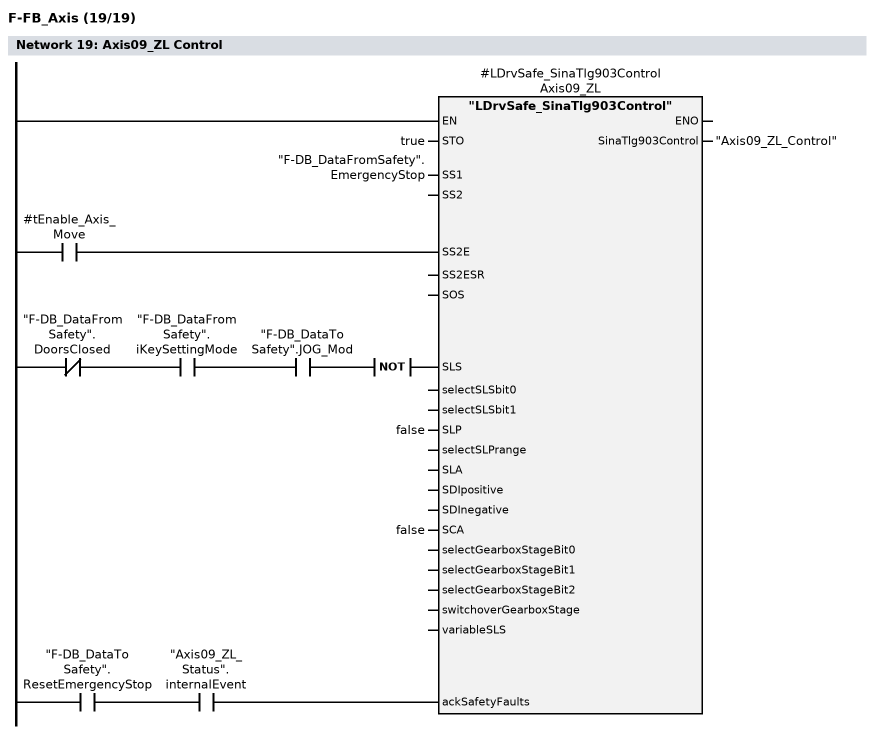
   RUNG wire#powerrail
      #LDrvSafe_SinaTlg903ControlAxis09_ZL(SS2E := wire#w1, SLS := wire#w2, ackSafetyFaults := wire#w3, STO := true, SS1 := "F-DB_DataFromSafety".EmergencyStop, SS2 :=, SS2ESR :=, SOS :=, selectSLSbit0 :=, selectSLSbit1 :=, SLP := false, selectSLPrange :=, SLA :=, SDIpositive :=, SDInegative :=, SCA := false, selectGearboxStageBit0 :=, selectGearboxStageBit1 :=, selectGearboxStageBit2 :=, switchoverGearboxStage :=, variableSLS :=, SinaTlg903Control => "Axis09_ZL_Control")
   END_RUNG
   RUNG wire#powerrail
      Contact( #tEnable_Axis_Move )
   END_RUNG wire#w1
   RUNG wire#powerrail
      I_Contact( "F-DB_DataFromSafety".DoorsClosed )
      Contact( "F-DB_DataFromSafety".iKeySettingMode )
      Contact( "F-DB_DataToSafety".JOG_Mod )
      Not()
   END_RUNG wire#w2
   RUNG wire#powerrail
      Contact( "F-DB_DataToSafety".ResetEmergencyStop )
      Contact( "Axis09_ZL_Status".internalEvent )
   END_RUNG wire#w3
   // the same network as SCL:
   #LDrvSafe_SinaTlg903ControlAxis09_ZL(STO := true,   // "LDrvSafe_SinaTlg903Control"
                           SS1 := "F-DB_DataFromSafety".EmergencyStop,
                           SS2E := #tEnable_Axis_Move,
                           SLS := NOT (NOT "F-DB_DataFromSafety".DoorsClosed AND "F-DB_DataFromSafety".iKeySettingMode AND "F-DB_DataToSafety".JOG_Mod),
                           SLP := false,
                           SCA := false,
                           ackSafetyFaults := "F-DB_DataToSafety".ResetEmergencyStop AND "Axis09_ZL_Status".internalEvent,
                           SinaTlg903Control => "Axis09_ZL_Control");
END_REGION
END_FUNCTION_BLOCK
